{attribute addProperty BoxType "EP2339-0042-0017"}
{attribute addProperty Id "DI_X01_Pin4AT %I*DI_X01_Pin_E4AEF59E810DI_X01_Pin2AT %I*DI_X01_Pin_E4AEF59E810DI_X02_Pin4AT %I*DI_X02_Pin_E4AEF59E810DI_X02_Pin2AT %I*DI_X02_Pin_E4AEF59E810DI_X03_Pin4AT %I*DI_X03_Pin_E4AEF59E810DI_X03_Pin2AT %I*DI_X03_Pin_E4AEF59E810DI_X04_Pin4AT %I*DI_X04_Pin_E4AEF59E810DI_X04_Pin2AT %I*DI_X04_Pin_E4AEF59E810DI_X05_Pin4AT %I*DI_X05_Pin_E4AEF59E810DI_X05_Pin2AT %I*DI_X05_Pin_E4AEF59E810DI_X06_Pin4AT %I*DI_X06_Pin_E4AEF59E810DI_X06_Pin2AT %I*DI_X06_Pin_E4AEF59E810DI_X07_Pin4AT %I*DI_X07_Pin_E4AEF59E810DI_X07_Pin2AT %I*DI_X07_Pin_E4AEF59E810DI_X08_Pin4AT %I*DI_X08_Pin_E4AEF59E810DI_X08_Pin2AT %I*DI_X08_Pin_E4AEF59E810DO_X01_PinAT %Q*ARRAY[0..1] OF DO_X01_Pin_7F374EB0429496728842949672950DO_X02_PinAT %Q*ARRAY[0..1] OF DO_X02_Pin_7F374EB0429496728842949672950DO_X03_PinAT %Q*ARRAY[0..1] OF DO_X03_Pin_7F374EB0429496728842949672950DO_X04_PinAT %Q*ARRAY[0..1] OF DO_X04_Pin_7F374EB0429496728842949672950DO_X05_PinAT %Q*ARRAY[0..1] OF DO_X05_Pin_7F374EB0429496728842949672950DO_X06_PinAT %Q*ARRAY[0..1] OF DO_X06_Pin_7F374EB0429496728842949672950DO_X07_PinAT %Q*ARRAY[0..1] OF DO_X07_Pin_7F374EB0429496728842949672950DO_X08_PinAT %Q*ARRAY[0..1] OF DO_X08_Pin_7F374EB0429496728842949672950WcStateAT %I*WcState_F855686C1620InfoDataAT %I*InfoData_192954DE1620"}
{attribute addProperty CRC "3801549111"}
{attribute addProperty SizeInBites "96"}
{attribute addProperty SizeInBytes "34359738380"}
TYPE EP2339_350240E0 :
STRUCT
	{attribute addProperty Name "DI_X01_Pin4"}
	DI_X01_Pin4 : DI_X01_Pin_E4AEF59E;
	{attribute addProperty Name "DI_X01_Pin2"}
	DI_X01_Pin2 : DI_X01_Pin_E4AEF59E;
	{attribute addProperty Name "DI_X02_Pin4"}
	DI_X02_Pin4 : DI_X02_Pin_E4AEF59E;
	{attribute addProperty Name "DI_X02_Pin2"}
	DI_X02_Pin2 : DI_X02_Pin_E4AEF59E;
	{attribute addProperty Name "DI_X03_Pin4"}
	DI_X03_Pin4 : DI_X03_Pin_E4AEF59E;
	{attribute addProperty Name "DI_X03_Pin2"}
	DI_X03_Pin2 : DI_X03_Pin_E4AEF59E;
	{attribute addProperty Name "DI_X04_Pin4"}
	DI_X04_Pin4 : DI_X04_Pin_E4AEF59E;
	{attribute addProperty Name "DI_X04_Pin2"}
	DI_X04_Pin2 : DI_X04_Pin_E4AEF59E;
	{attribute addProperty Name "DI_X05_Pin4"}
	DI_X05_Pin4 : DI_X05_Pin_E4AEF59E;
	{attribute addProperty Name "DI_X05_Pin2"}
	DI_X05_Pin2 : DI_X05_Pin_E4AEF59E;
	{attribute addProperty Name "DI_X06_Pin4"}
	DI_X06_Pin4 : DI_X06_Pin_E4AEF59E;
	{attribute addProperty Name "DI_X06_Pin2"}
	DI_X06_Pin2 : DI_X06_Pin_E4AEF59E;
	{attribute addProperty Name "DI_X07_Pin4"}
	DI_X07_Pin4 : DI_X07_Pin_E4AEF59E;
	{attribute addProperty Name "DI_X07_Pin2"}
	DI_X07_Pin2 : DI_X07_Pin_E4AEF59E;
	{attribute addProperty Name "DI_X08_Pin4"}
	DI_X08_Pin4 : DI_X08_Pin_E4AEF59E;
	{attribute addProperty Name "DI_X08_Pin2"}
	DI_X08_Pin2 : DI_X08_Pin_E4AEF59E;
	{attribute addProperty Name "DO_X01_Pin"}
	DO_X01_Pin : ARRAY[0..1] OF DO_X01_Pin_7F374EB0;
	{attribute addProperty Name "DO_X02_Pin"}
	DO_X02_Pin : ARRAY[0..1] OF DO_X02_Pin_7F374EB0;
	{attribute addProperty Name "DO_X03_Pin"}
	DO_X03_Pin : ARRAY[0..1] OF DO_X03_Pin_7F374EB0;
	{attribute addProperty Name "DO_X04_Pin"}
	DO_X04_Pin : ARRAY[0..1] OF DO_X04_Pin_7F374EB0;
	{attribute addProperty Name "DO_X05_Pin"}
	DO_X05_Pin : ARRAY[0..1] OF DO_X05_Pin_7F374EB0;
	{attribute addProperty Name "DO_X06_Pin"}
	DO_X06_Pin : ARRAY[0..1] OF DO_X06_Pin_7F374EB0;
	{attribute addProperty Name "DO_X07_Pin"}
	DO_X07_Pin : ARRAY[0..1] OF DO_X07_Pin_7F374EB0;
	{attribute addProperty Name "DO_X08_Pin"}
	DO_X08_Pin : ARRAY[0..1] OF DO_X08_Pin_7F374EB0;
	{attribute addProperty Name "WcState"}
	WcState : WcState_F855686C;
	{attribute addProperty Name "InfoData"}
	InfoData : InfoData_192954DE;
END_STRUCT
END_TYPE

(* stored: Version 1.2.0.0, ProductVersion 3.1.4024.9
   DUT EP2339_350240E0: Id {a8e269d6-11ac-459e-af1a-2814f68a654f} *)
